// TIA Portal V19 export
VAR_GLOBAL   // PLC tag table "Default tag table"
   start AT %I0.0 : Bool;
   stop AT %I0.1 : Bool;
   L1 AT %Q0.0 : Bool;
END_VAR
